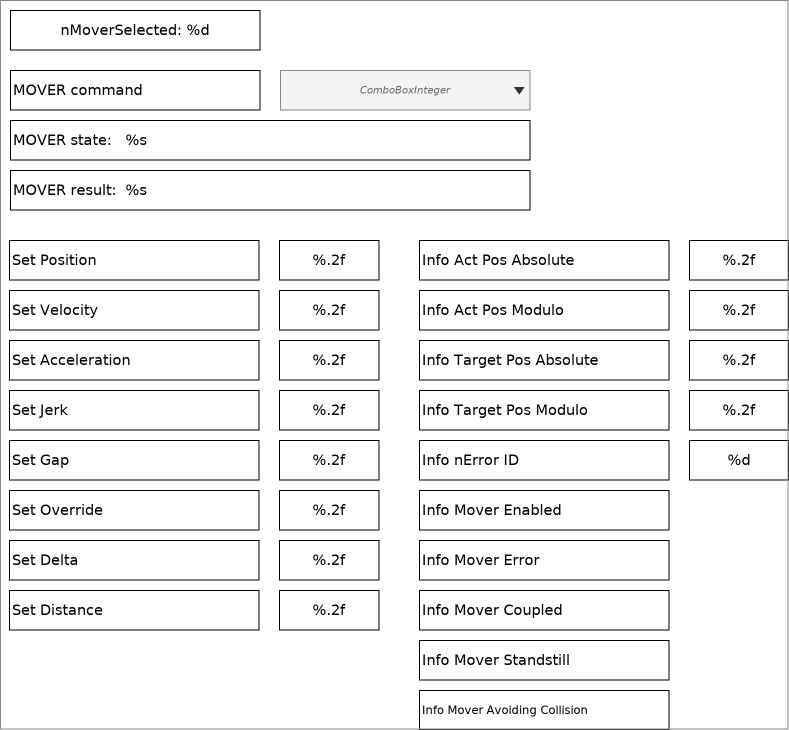
VISUALIZATION MOVER_VISU  // 789x730
    Rectangle (10,10 250x40), "nMoverSelected: %d", text variable: MAIN.nMoverSelected
        OnMouseClick: write the text variable via VisuDialogs.Numpad, min 1, max MAX_MOVER, title 'Selected Mover'
    Rectangle (10,120 520x40), "MOVER state: %s", text variable: MAIN.sMoverState
    Rectangle (10,70 250x40), "MOVER command"
    ComboBoxInteger (280,70 250x40), variable: GVL_XTS.MoverCtrl[MAIN.nMoverSelected].Cmd, text list: 'TL_E_CTRL_MOVER'
    Rectangle (10,170 520x40), "MOVER result: %s", text variable: MAIN.sMoverResult
    Rectangle (9,240 250x40), "Set Position"
    Rectangle (9,290 250x40), "Set Velocity"
    Rectangle (9,340 250x40), "Set Acceleration"
    Rectangle (9,390 250x40), "Set Jerk"
    Rectangle (9,440 250x40), "Set Gap"
    Rectangle (9,490 250x40), "Set Override"
    Rectangle (9,540 250x40), "Set Delta"
    Rectangle (9,590 250x40), "Set Distance"
    Rectangle (279,240 100x40), "%.2f", text variable: GVL_XTS.MoveData[MAIN.nMoverSelected].rPos
        OnMouseClick: write the text variable via Default
    Rectangle (279,290 100x40), "%.2f", text variable: GVL_XTS.MoveData[MAIN.nMoverSelected].rVelo
        OnMouseClick: write the text variable via Default
    Rectangle (279,340 100x40), "%.2f", text variable: GVL_XTS.MoveData[MAIN.nMoverSelected].rAcc
        OnMouseClick: write the text variable via Default
    Rectangle (279,390 100x40), "%.2f", text variable: GVL_XTS.MoveData[MAIN.nMoverSelected].rJerk
        OnMouseClick: write the text variable via Default
    Rectangle (279,440 100x40), "%.2f", text variable: GVL_XTS.MoveData[MAIN.nMoverSelected].rGap
        OnMouseClick: write the text variable via Default
    Rectangle (279,490 100x40), "%.2f", text variable: GVL_XTS.MoveData[MAIN.nMoverSelected].rOverride
        OnMouseClick: write the text variable via Default
    Rectangle (279,540 100x40), "%.2f", text variable: GVL_XTS.MoveData[MAIN.nMoverSelected].rDelta
        OnMouseClick: write the text variable via Default
    Rectangle (279,590 100x40), "%.2f", text variable: GVL_XTS.MoveData[MAIN.nMoverSelected].rDistance
        OnMouseClick: write the text variable via Default
    Rectangle (419,240 250x40), "Info Act Pos Absolute"
    Rectangle (419,290 250x40), "Info Act Pos Modulo"
    Rectangle (419,340 250x40), "Info Target Pos Absolute"
    Rectangle (419,390 250x40), "Info Target Pos Modulo"
    Rectangle (419,440 250x40), "Info nError ID"
    Rectangle (689,240 100x40), "%.2f", text variable: GVL_XTS.MoverInfo[MAIN.nMoverSelected].rAbsActPos
    Rectangle (689,290 100x40), "%.2f", text variable: GVL_XTS.MoverInfo[MAIN.nMoverSelected].rModuloActPos
    Rectangle (689,340 100x40), "%.2f", text variable: GVL_XTS.MoverInfo[MAIN.nMoverSelected].rAbsTargetPos
    Rectangle (689,390 100x40), "%.2f", text variable: GVL_XTS.MoverInfo[MAIN.nMoverSelected].rModuloTargetPos
    Rectangle (689,440 100x40), "%d", text variable: GVL_XTS.MoverInfo[MAIN.nMoverSelected].nErrorId
    Rectangle (419,490 250x40), "Info Mover Enabled", colour toggle: GVL_XTS.MoverInfo[MAIN.nMoverSelected].bMoverEnabled
    Rectangle (419,540 250x40), "Info Mover Error", colour toggle: GVL_XTS.MoverInfo[MAIN.nMoverSelected].bMoverError
    Rectangle (419,590 250x40), "Info Mover Coupled", colour toggle: GVL_XTS.MoverInfo[MAIN.nMoverSelected].bMoverCoupled
    Rectangle (419,640 250x40), "Info Mover Standstill", colour toggle: GVL_XTS.MoverInfo[MAIN.nMoverSelected].bMoverStandstill
    Rectangle (419,690 250x40), "Info Mover Avoiding Collision", colour toggle: GVL_XTS.MoverInfo[MAIN.nMoverSelected].bMoverAvoidingCollision
END_VISUALIZATION

(* stored: Version 1.1.0.1
   Visu MOVER_VISU: Id {c9fb373c-2482-41b3-8168-553de4317393} *)
